(* IEC 61131-3 sources: RL_MAR/experiments/comparison/autoplc/results/gpt-4o-mini_20260511_164212/med_45, 1 file *)

(* ---- med_45_1.st ---- *)
FUNCTION_BLOCK AutomatedSmoothieMaker
    VAR_INPUT
        BananaAvailable : BOOL;
        BerryMixAvailable : BOOL;
        SpinachAvailable : BOOL;
        YogurtAvailable : BOOL;
        CustomerPreference : INT;
    END_VAR

    VAR_OUTPUT
        BlenderMotor : BOOL := FALSE;
        Dispenser : BOOL := FALSE;
    END_VAR

    VAR
        RecipeValid : BOOL := FALSE;
        IngredientsAvailable : BOOL := FALSE;
    END_VAR

    // Check customer preference and ingredient availability
    IF CustomerPreference >= 1 AND CustomerPreference <= 3 THEN
        RecipeValid := TRUE;

        CASE CustomerPreference OF
            1: // Recipe 1: Banana, Berry Mix, Yogurt
                IngredientsAvailable := BananaAvailable AND BerryMixAvailable AND YogurtAvailable;
            2: // Recipe 2: Berry Mix, Spinach, Yogurt
                IngredientsAvailable := BerryMixAvailable AND SpinachAvailable AND YogurtAvailable;
            3: // Recipe 3: Banana, Spinach, Yogurt
                IngredientsAvailable := BananaAvailable AND SpinachAvailable AND YogurtAvailable;
            ELSE
                RecipeValid := FALSE; // Invalid preference
        END_CASE
    ELSE
        RecipeValid := FALSE; // Invalid preference
    END_IF

    // Control logic based on availability and preference
    IF RecipeValid AND IngredientsAvailable THEN
        // Start blending process
        BlenderMotor := TRUE;
        Dispenser := TRUE;
    ELSE
        // Turn off blender and dispenser in case of error
        BlenderMotor := FALSE;
        Dispenser := FALSE;
    END_IF

    // Simulate blending process duration (for example, using a simple delay or counter)
    // Here we assume blending takes place for a fixed duration
    // This part can be replaced with actual timing logic if needed
    // For demonstration, we will just turn off after one cycle
    IF BlenderMotor THEN
        // After blending, turn off the motor and dispenser
        BlenderMotor := FALSE;
        Dispenser := FALSE;
    END_IF

END_FUNCTION_BLOCK
